// TIA Portal V16 export
// export: Created 2021-09-08T12:46:16.1780561Z, ExportSetting WithDefaults, DisplayName Totally Integrated Automation Portal, DisplayVersion V16 Update 3, DisplayName TIA Portal Version Control Interface, DisplayVersion V16 Update 2, DisplayName TIA Portal Openness, DisplayVersion V16 Update 3, DisplayName TIA Portal Teamcenter Gateway, DisplayVersion V16, DisplayName STEP 7 Professional, DisplayVersion V16 Update 3, DisplayName STEP 7 Safety, DisplayVersion V16, DisplayName WinCC Advanced, DisplayVersion V16 Update 3
TYPE "FREQ_COUNTER"
// stored: IsFailsafeCompliant false
   STRUCT
      litrsPerPuls : UInt;
      prewHour : UInt;
      curHour : UInt;
      prewDay : UDInt;
      curDay : UDInt;
      all : UDInt;
      rst : Bool;
   END_STRUCT;
END_TYPE
